(* PLC project Plc, Beckhoff Automation GmbH TwinCAT PLC Control 3.5.20.60 *)
(* stored: creationDateTime 2025-11-03T13:47:02.2969609, modificationDateTime 2025-11-03T13:47:02.3009785 *)

FUNCTION_BLOCK FB_VarByteBuffer IMPLEMENTS I_VarByteBuffer
VAR
	_pBuffer 	: POINTER TO BYTE;
	_nHead 		: UDINT;
	_nCapacity 	: UDINT;
	
	_nError : UDINT;
END_VAR
VAR CONSTANT
	cMaxBufferSize 		: UDINT := 104857600 ; // 100 Mb
END_VAR

            
          

//FB_Exit must be implemented explicitly. If there is an implementation, then the
//method is called before the controller removes the code of the function block instance
//(implicit call). The return value is not evaluated.
METHOD FB_Exit: BOOL
VAR_INPUT
    bInCopyCode: BOOL;  // TRUE: the exit method is called in order to leave the instance which will be copied afterwards (online change).  
END_VAR
                  this^.Reset();
                
END_METHOD

METHOD Initialize : BOOL
VAR_INPUT
	nBufferSize 		: UDINT; // Size in byte
END_VAR
                  IF nBufferSize = 0 OR nBufferSize > THIS^.cMaxBufferSize THEN RETURN; END_IF;

THIS^.Reset();

THIS^._nCapacity := nBufferSize;
THIS^._pBuffer := __NEW(BYTE, nBufferSize);
IF THIS^._pBuffer = 0 THEN RETURN; END_IF;

Initialize := TRUE;
                
END_METHOD

METHOD Push : BOOL
VAR_INPUT
	pData : pvoid;
	cbSize : UDINT;
END_VAR
VAR;
	res			: UDINT;
END_VAR
                  IF (THIS^._pBuffer = 0) OR (THIS^._nCapacity = 0) THEN RETURN; END_IF;		// Check initialization
IF pData = 0 THEN RETURN; END_IF											// Check input
IF THIS^.FreeBytes < cbSize THEN RETURN; END_IF;

res := memcpy(THIS^._pBuffer + THIS^._nHead,pData,cbSize);
IF res <> cbSize THEN
	THIS^._nError := THIS^._nError + 1; 
	RETURN;
END_IF

THIS^._nHead := THIS^._nHead + cbSize;

Push := TRUE;
                
END_METHOD

METHOD Reset
                  IF THIS^._pBuffer <> 0 THEN
	__DELETE(THIS^._pBuffer);
	THIS^._pBuffer := 0;
END_IF

THIS^._nHead 			:= 0;
THIS^._nCapacity 		:= 0;
THIS^._nError 			:= 0;
                
END_METHOD

METHOD Clear : BOOL
VAR
	res : UDINT;
END_VAR
                  res := memset(THIS^.Buffer, 0, THIS^.Capacity);
IF res <> THIS^.Capacity THEN RETURN; END_IF
THIS^._nHead := 0;
Clear := true;
                
END_METHOD

PROPERTY Capacity : UDINT
GET
VAR
END_VAR
                    Capacity := this^._nCapacity;
                  
END_GET
END_PROPERTY

PROPERTY Size : UDINT
GET
VAR
END_VAR
                    Size := this^._nHead;
                  
END_GET
END_PROPERTY

PROPERTY Buffer : PVOID
GET
VAR
END_VAR
                    Buffer := THIS^._pBuffer;
                  
END_GET
END_PROPERTY

PROPERTY FreeBytes : UDINT
GET
VAR
END_VAR
                    FreeBytes := THIS^._nCapacity - this^._nHead;
                  
END_GET
END_PROPERTY
END_FUNCTION_BLOCK
